# B&R Automation Studio project Servo
Automation Studio 4.12.2.93; technology packages: mappMotion 5.23.1, mappView 5.23.0

## Configuration Config1

CPU X20CP1586, AutomationRuntime B4.93, Build 4.1.2, Vc V4.72.6

### Task classes (Cpu.sw)
```
Cyclic#1 (cycle 8000 us, tolerance 0 us):
  servo <- servo.prg
DataObjects: McAcpSys
NcDataObjects: McDriveLog
Binaries: FWRules, McAcpSim, arcoal, arsvcreg, TCData, McAcpDrv, arflatprv, udbdef, iomap, Config_1, ashwd, arconfig, asfw, ashwac, sysconf, User, Role
Libraries: McBase, MpAxis, McAxis, MpBase, McAcpAx, fileio, powerlnk, sys_lib, asieccon, asepl, standard, MpAlarmX, astime, runtime
```

### Hardware
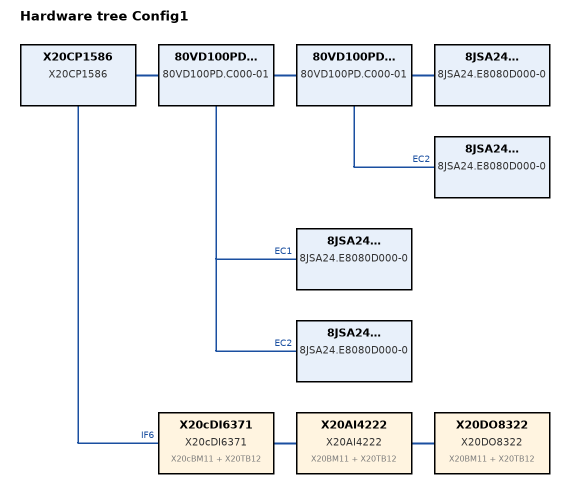
```
80VD100PD.C000-01 : 80VD100PD.C000-01 v2.5.0.0  [PLK1 -> 80VD100PD.C000-01a.PLK2 (NodeNumber=2) [Cable Type=PowerlinkCable, Length=10, Version=1.0.0.3]; EC1 -> 8JSA24.E8080D000-0.EC; EC2 -> 8JSA24.E8080D000-0a.EC; MT2 -> 8JSA24.E8080D000-0a.MT]
  DriveConfiguration/Module:
    McAcoposTypeID = AcoposMicroDConfig
    ActivateACOPOSSimulationOnPLC = 1
  DriveConfiguration/Channel[1]/RealAxis:
    AxisReference = gAxis_1
    MechanicalElementsIsInvisible = 0
  DriveConfiguration/Channel[1]/RealAxis/MechanicalElements/Gearbox:
    InputIsReadOnly = 0
    Input = 1
    OutputIsReadOnly = 0
    Output = 1
  DriveConfiguration/Channel[1]/RealAxis/MechanicalElements/RotaryToLinearTransformation:
    ReferenceDistanceIsReadOnly = 0
    ReferenceDistance = 1
  DriveConfiguration/Channel[1]/RealAxis/Controller:
    ModeIsReadOnly = 0
    Mode = PositionController
  DriveConfiguration/Channel[1]/RealAxis/Controller/Mode/Position:
    ProportionalGain = 50.0
    IntegrationTime = 0.0
    PredictionTime = 0.0004
    TotalDelayTime = 0.0004
  DriveConfiguration/Channel[1]/RealAxis/Controller/Mode/Speed:
    ProportionalGainIsReadOnly = 0
    ProportionalGain = 2.0
    IntegrationTimeIsReadOnly = 0
    IntegrationTime = 0.0
    FilterTimeIsReadOnly = 0
    FilterTime = 0.0
  DriveConfiguration/Channel[1]/RealAxis/Controller/Mode/LoopFilters:
    LoopFilterXIsReadOnly = 0
    LoopFilter1 = NotUsed
    LoopFilter2 = NotUsed
    LoopFilter3 = NotUsed
  DriveConfiguration/Channel[1]/RealAxis/Homing:
    ModeIsReadOnly = 0
    Mode = Direct
  DriveConfiguration/Channel[1]/RealAxis/Homing/Mode:
    Position = 0.0
    ReferencePulse = NotUsed
  DriveConfiguration/Channel[1]/RealAxis/Homing:
    RestorePositionVariable = 
  DriveConfiguration/Channel[1]/RealAxis/StopReaction:
    QuickstopIsReadOnly = 0
    Quickstop = DecelerationLimit
    DriveErrorIsReadOnly = 0
    DriveError = DecelerationLimit
  DriveConfiguration/Channel[1]/RealAxis/MovementErrorLimits:
    PositionError = 1.0
    VelocityErrorMonitoring = Automatic1
  DriveConfiguration/Channel[1]/RealAxis:
    JerkFilterIsReadOnly = 0
    JerkFilter = NotUsed
    ZeroVibrationFilter = NotUsed
  DriveConfiguration/Channel[1]/RealAxis/DigitalInputs/HomingSwitch:
    SourceIsReadOnly = 0
    Source = NotUsed
    Level = High
  DriveConfiguration/Channel[1]/RealAxis/DigitalInputs/PositiveLimitSwitch:
    SourceIsReadOnly = 0
    Source = NotUsed
    Level = High
  DriveConfiguration/Channel[1]/RealAxis/DigitalInputs/NegativeLimitSwitch:
    SourceIsReadOnly = 0
    Source = NotUsed
    Level = High
  DriveConfiguration/Channel[1]/RealAxis/DigitalInputs/Trigger1:
    Source = X2Trigger1
    Level = High
  DriveConfiguration/Channel[1]/RealAxis/DigitalInputs/Trigger2:
    Source = X2Trigger2
    Level = High
  DriveConfiguration/Channel[1]/RealAxis/DigitalInputs/Quickstop:
    Input = Trigger2
  DriveConfiguration/Channel[1]/RealAxis/Simulation:
    SimulationModeOnPLC = SetValueGeneration
    SimulationModeOnACOPOS = NotUsed
  DriveConfiguration/Channel[2]/RealAxis:
    AxisReference = gAxis_2
    MechanicalElementsIsInvisible = 0
  DriveConfiguration/Channel[2]/RealAxis/MechanicalElements/Gearbox:
    InputIsReadOnly = 0
    Input = 1
    OutputIsReadOnly = 0
    Output = 1
  DriveConfiguration/Channel[2]/RealAxis/MechanicalElements/RotaryToLinearTransformation:
    ReferenceDistanceIsReadOnly = 0
    ReferenceDistance = 1
  DriveConfiguration/Channel[2]/RealAxis/Controller:
    ModeIsReadOnly = 0
    Mode = PositionController
  DriveConfiguration/Channel[2]/RealAxis/Controller/Mode/Position:
    ProportionalGain = 50.0
    IntegrationTime = 0.0
    PredictionTime = 0.0004
    TotalDelayTime = 0.0004
  DriveConfiguration/Channel[2]/RealAxis/Controller/Mode/Speed:
    ProportionalGainIsReadOnly = 0
    ProportionalGain = 2.0
    IntegrationTimeIsReadOnly = 0
    IntegrationTime = 0.0
    FilterTimeIsReadOnly = 0
    FilterTime = 0.0
  DriveConfiguration/Channel[2]/RealAxis/Controller/Mode/LoopFilters:
    LoopFilterXIsReadOnly = 0
    LoopFilter1 = NotUsed
    LoopFilter2 = NotUsed
    LoopFilter3 = NotUsed
  DriveConfiguration/Channel[2]/RealAxis/Homing:
    ModeIsReadOnly = 0
    Mode = Direct
  DriveConfiguration/Channel[2]/RealAxis/Homing/Mode:
    Position = 0.0
    ReferencePulse = NotUsed
  DriveConfiguration/Channel[2]/RealAxis/Homing:
    RestorePositionVariable = 
  DriveConfiguration/Channel[2]/RealAxis/StopReaction:
    QuickstopIsReadOnly = 0
    Quickstop = DecelerationLimit
    DriveErrorIsReadOnly = 0
    DriveError = DecelerationLimit
  DriveConfiguration/Channel[2]/RealAxis/MovementErrorLimits:
    PositionError = 1.0
    VelocityErrorMonitoring = Automatic1
  DriveConfiguration/Channel[2]/RealAxis:
    JerkFilterIsReadOnly = 0
    JerkFilter = NotUsed
    ZeroVibrationFilter = NotUsed
  DriveConfiguration/Channel[2]/RealAxis/DigitalInputs/HomingSwitch:
    SourceIsReadOnly = 0
    Source = NotUsed
    Level = High
  DriveConfiguration/Channel[2]/RealAxis/DigitalInputs/PositiveLimitSwitch:
    SourceIsReadOnly = 0
    Source = NotUsed
    Level = High
  DriveConfiguration/Channel[2]/RealAxis/DigitalInputs/NegativeLimitSwitch:
    SourceIsReadOnly = 0
    Source = NotUsed
    Level = High
  DriveConfiguration/Channel[2]/RealAxis/DigitalInputs/Trigger1:
    Source = X2Trigger1
    Level = High
  DriveConfiguration/Channel[2]/RealAxis/DigitalInputs/Trigger2:
    Source = X2Trigger2
    Level = High
  DriveConfiguration/Channel[2]/RealAxis/DigitalInputs/Quickstop:
    Input = Trigger2
  DriveConfiguration/Channel[2]/RealAxis/Simulation:
    SimulationModeOnPLC = SetValueGeneration
    SimulationModeOnACOPOS = NotUsed
80VD100PD.C000-01a : 80VD100PD.C000-01 v2.5.0.0  [PLK1 -> X20CP1586.IF3 (NodeNumber=3) [Cable Type=PowerlinkCable, Length=10, Version=1.0.0.3]; PLK2 -> 80VD100PD.C000-01.PLK1 (NodeNumber=3) [Cable Type=PowerlinkCable, Length=10, Version=1.0.0.3]; EC1 -> 8JSA24.E8080D000-0b.EC; EC2 -> 8JSA24.E8080D000-0c.EC; MT2 -> 8JSA24.E8080D000-0c.MT]
  DriveConfiguration/Module:
    McAcoposTypeID = AcoposMicroDConfig
    ActivateACOPOSSimulationOnPLC = 1
  DriveConfiguration/Channel[1]/RealAxis:
    AxisReference = gAxis_3
    MechanicalElementsIsInvisible = 0
  DriveConfiguration/Channel[1]/RealAxis/MechanicalElements/Gearbox:
    InputIsReadOnly = 0
    Input = 1
    OutputIsReadOnly = 0
    Output = 1
  DriveConfiguration/Channel[1]/RealAxis/MechanicalElements/RotaryToLinearTransformation:
    ReferenceDistanceIsReadOnly = 0
    ReferenceDistance = 1
  DriveConfiguration/Channel[1]/RealAxis/Controller:
    ModeIsReadOnly = 0
    Mode = PositionController
  DriveConfiguration/Channel[1]/RealAxis/Controller/Mode/Position:
    ProportionalGain = 50.0
    IntegrationTime = 0.0
    PredictionTime = 0.0004
    TotalDelayTime = 0.0004
  DriveConfiguration/Channel[1]/RealAxis/Controller/Mode/Speed:
    ProportionalGainIsReadOnly = 0
    ProportionalGain = 2.0
    IntegrationTimeIsReadOnly = 0
    IntegrationTime = 0.0
    FilterTimeIsReadOnly = 0
    FilterTime = 0.0
  DriveConfiguration/Channel[1]/RealAxis/Controller/Mode/LoopFilters:
    LoopFilterXIsReadOnly = 0
    LoopFilter1 = NotUsed
    LoopFilter2 = NotUsed
    LoopFilter3 = NotUsed
  DriveConfiguration/Channel[1]/RealAxis/Homing:
    ModeIsReadOnly = 0
    Mode = Direct
  DriveConfiguration/Channel[1]/RealAxis/Homing/Mode:
    Position = 0.0
    ReferencePulse = Used
  DriveConfiguration/Channel[1]/RealAxis/Homing/Mode/ReferencePulse:
    HomingVelocity = 0.5
    Acceleration = 50.0
    HomingDirection = Positive
    KeepDirection = No
    ReferencePulseBlockingDistance = 0.0
  DriveConfiguration/Channel[1]/RealAxis/Homing:
    RestorePositionVariable = 
  DriveConfiguration/Channel[1]/RealAxis/StopReaction:
    QuickstopIsReadOnly = 0
    Quickstop = DecelerationLimit
    DriveErrorIsReadOnly = 0
    DriveError = DecelerationLimit
  DriveConfiguration/Channel[1]/RealAxis/MovementErrorLimits:
    PositionError = 1.0
    VelocityErrorMonitoring = Automatic1
  DriveConfiguration/Channel[1]/RealAxis:
    JerkFilterIsReadOnly = 0
    JerkFilter = NotUsed
    ZeroVibrationFilter = NotUsed
  DriveConfiguration/Channel[1]/RealAxis/DigitalInputs/HomingSwitch:
    SourceIsReadOnly = 0
    Source = NotUsed
    Level = High
  DriveConfiguration/Channel[1]/RealAxis/DigitalInputs/PositiveLimitSwitch:
    SourceIsReadOnly = 0
    Source = NotUsed
    Level = High
  DriveConfiguration/Channel[1]/RealAxis/DigitalInputs/NegativeLimitSwitch:
    SourceIsReadOnly = 0
    Source = NotUsed
    Level = High
  DriveConfiguration/Channel[1]/RealAxis/DigitalInputs/Trigger1:
    Source = X2Trigger1
    Level = High
  DriveConfiguration/Channel[1]/RealAxis/DigitalInputs/Trigger2:
    Source = X2Trigger2
    Level = High
  DriveConfiguration/Channel[1]/RealAxis/DigitalInputs/Quickstop:
    Input = Trigger2
  DriveConfiguration/Channel[1]/RealAxis/Simulation:
    SimulationModeOnPLC = SetValueGeneration
    SimulationModeOnACOPOS = NotUsed
  DriveConfiguration/Channel[2]/RealAxis:
    AxisReference = gAxis_4
    MechanicalElementsIsInvisible = 0
  DriveConfiguration/Channel[2]/RealAxis/MechanicalElements/Gearbox:
    InputIsReadOnly = 0
    Input = 1
    OutputIsReadOnly = 0
    Output = 1
  DriveConfiguration/Channel[2]/RealAxis/MechanicalElements/RotaryToLinearTransformation:
    ReferenceDistanceIsReadOnly = 0
    ReferenceDistance = 1
  DriveConfiguration/Channel[2]/RealAxis/Controller:
    ModeIsReadOnly = 0
    Mode = PositionController
  DriveConfiguration/Channel[2]/RealAxis/Controller/Mode/Position:
    ProportionalGain = 50.0
    IntegrationTime = 0.0
    PredictionTime = 0.0004
    TotalDelayTime = 0.0004
  DriveConfiguration/Channel[2]/RealAxis/Controller/Mode/Speed:
    ProportionalGainIsReadOnly = 0
    ProportionalGain = 2.0
    IntegrationTimeIsReadOnly = 0
    IntegrationTime = 0.0
    FilterTimeIsReadOnly = 0
    FilterTime = 0.0
  DriveConfiguration/Channel[2]/RealAxis/Controller/Mode/LoopFilters:
    LoopFilterXIsReadOnly = 0
    LoopFilter1 = NotUsed
    LoopFilter2 = NotUsed
    LoopFilter3 = NotUsed
  DriveConfiguration/Channel[2]/RealAxis/Homing:
    ModeIsReadOnly = 0
    Mode = Direct
  DriveConfiguration/Channel[2]/RealAxis/Homing/Mode:
    Position = 0.0
    ReferencePulse = NotUsed
  DriveConfiguration/Channel[2]/RealAxis/Homing:
    RestorePositionVariable = 
  DriveConfiguration/Channel[2]/RealAxis/StopReaction:
    QuickstopIsReadOnly = 0
    Quickstop = DecelerationLimit
    DriveErrorIsReadOnly = 0
    DriveError = DecelerationLimit
  DriveConfiguration/Channel[2]/RealAxis/MovementErrorLimits:
    PositionError = 1.0
    VelocityErrorMonitoring = Automatic1
  DriveConfiguration/Channel[2]/RealAxis:
    JerkFilterIsReadOnly = 0
    JerkFilter = NotUsed
    ZeroVibrationFilter = NotUsed
  DriveConfiguration/Channel[2]/RealAxis/DigitalInputs/HomingSwitch:
    SourceIsReadOnly = 0
    Source = NotUsed
    Level = High
  DriveConfiguration/Channel[2]/RealAxis/DigitalInputs/PositiveLimitSwitch:
    SourceIsReadOnly = 0
    Source = NotUsed
    Level = High
  DriveConfiguration/Channel[2]/RealAxis/DigitalInputs/NegativeLimitSwitch:
    SourceIsReadOnly = 0
    Source = NotUsed
    Level = High
  DriveConfiguration/Channel[2]/RealAxis/DigitalInputs/Trigger1:
    Source = X2Trigger1
    Level = High
  DriveConfiguration/Channel[2]/RealAxis/DigitalInputs/Trigger2:
    Source = X2Trigger2
    Level = High
  DriveConfiguration/Channel[2]/RealAxis/DigitalInputs/Quickstop:
    Input = Trigger2
  DriveConfiguration/Channel[2]/RealAxis/Simulation:
    SimulationModeOnPLC = SetValueGeneration
    SimulationModeOnACOPOS = NotUsed
8JSA24.E8080D000-0 : 8JSA24.E8080D000-0 v1.0.6.30  [EC -> 80VD100PD.C000-01.EC1; MT -> 80VD100PD.C000-01.MT1]
8JSA24.E8080D000-0a : 8JSA24.E8080D000-0 v1.0.6.30  [EC -> 80VD100PD.C000-01.EC2; MT -> 80VD100PD.C000-01.MT2]
8JSA24.E8080D000-0b : 8JSA24.E8080D000-0 v1.0.6.30  [EC -> 80VD100PD.C000-01a.EC1; MT -> 80VD100PD.C000-01a.MT1]
8JSA24.E8080D000-0c : 8JSA24.E8080D000-0 v1.0.6.30  [EC -> 80VD100PD.C000-01a.EC2; MT -> 80VD100PD.C000-01a.MT2]
X20AI4222 : X20AI4222 v1.2.0.0  [SS1 -> X20TB12b.SS; SL -> X20BM11a.SL1]
X20BM11 : X20BM11 v1.1.0.0  [X2X1 -> X20BM11a.X2X2]
X20BM11a : X20BM11 v1.1.0.0  [X2X1 -> X20cBM11.X2X2]
X20CP1586 : X20CP1586 v1.10.0.0
  Connector IF2:
    ActivateDevice = 1
  ConfigurationID = Servo_Config1
  Simulation = 1
  TimerDeviceType = EPLX2X
  TimerDevice = X20CP1586.IF3
  TaskClassIdleTime = 2000
  Cyclic1Duration = 8000
  Cyclic1Tolerance = 0
  Cyclic1Stack = 35563
  FileDevice1
  FileDeviceName1 = USER
  FileDevicePath1 = USER_PATH
  ActivateOpcUa = 1
  OpcUaInformationModels_PV_Version = 1
X20DO8322 : X20DO8322 v1.5.0.0  [SS1 -> X20TB12a.SS; SL -> X20BM11.SL1]
X20TB12 : X20TB12 v1.0.0.0
X20TB12a : X20TB12 v1.0.0.0
X20TB12b : X20TB12 v1.0.0.0
X20cBM11 : X20cBM11 v1.1.0.0  [X2X1 -> X20CP1586.IF6]
X20cDI6371 : X20cDI6371 v1.2.0.0  [SS1 -> X20TB12.SS; SL -> X20cBM11.SL1]
```

### IoMap.iom - X20CP1586/IoMap.iom
```iecst
VAR_CONFIG
	::KEY AT %IX."X20cDI6371".DigitalInput01;
	::Left_Proximity AT %IX."X20cDI6371".DigitalInput03;
	::Buzzer AT %QX."X20DO8322".DigitalOutput01;
	::LeftAct AT %QX."X20DO8322".DigitalOutput02;
	::RightAct AT %QX."X20DO8322".DigitalOutput03;
	::Proximity_1 AT %IX."X20cDI6371".DigitalInput02;
	::Right_Proximity AT %IX."X20cDI6371".DigitalInput04;
END_VAR
```

### Config_1.axis - X20CP1586/mappMotion/Config_1.axis
```
Element gAxis_1 (Type=axis)
  BaseTypeIsReadOnly = 0
  BaseType = LinearBounded
    MeasurementUnit = 5066068
    MeasurementResolutionIsReadOnly = 0
    MeasurementResolution = 0.01
    CountDirectionIsReadOnly = 0
    CountDirection = Standard
  MovementLimitsIsReadOnly = 0
  MovementLimits = Internal
    Position:
      LowerLimitMin = -1.79769313486231E308
      UpperLimitMax = 1.79769313486231E308
      LowerLimit = -100000
      UpperLimit = 100000
    VelocityIsReadOnly = 0
    Velocity:
      VelocityMax = 3.4E38
      Velocity = 10
    AccelerationIsReadOnly = 0
    Acceleration:
      AccelerationMax = 3.4E38
      Acceleration = 50
    DecelerationIsReadOnly = 0
    Deceleration:
      DecelerationMax = 3.4E38
      Deceleration = 50.0
  Alarms = None
```

### Config_2.axis - X20CP1586/mappMotion/Config_2.axis
```
Element gAxis_2 (Type=axis)
  BaseTypeIsReadOnly = 0
  BaseType = LinearBounded
    MeasurementUnit = 5066068
    MeasurementResolutionIsReadOnly = 0
    MeasurementResolution = 0.01
    CountDirectionIsReadOnly = 0
    CountDirection = Standard
  MovementLimitsIsReadOnly = 0
  MovementLimits = Internal
    Position:
      LowerLimitMin = -1.79769313486231E308
      UpperLimitMax = 1.79769313486231E308
      LowerLimit = -1000.0
      UpperLimit = 1000.0
    VelocityIsReadOnly = 0
    Velocity:
      VelocityMax = 3.4E38
      Velocity = 10.0
    AccelerationIsReadOnly = 0
    Acceleration:
      AccelerationMax = 3.4E38
      Acceleration = 50.0
    DecelerationIsReadOnly = 0
    Deceleration:
      DecelerationMax = 3.4E38
      Deceleration = 50.0
  Alarms = None
```

### Config_3.axis - X20CP1586/mappMotion/Config_3.axis
```
Element gAxis_3 (Type=axis)
  BaseTypeIsReadOnly = 0
  BaseType = LinearBounded
    MeasurementUnit = 5066068
    MeasurementResolutionIsReadOnly = 0
    MeasurementResolution = 0.01
    CountDirectionIsReadOnly = 0
    CountDirection = Standard
  MovementLimitsIsReadOnly = 0
  MovementLimits = Internal
    Position:
      LowerLimitMin = -1.79769313486231E308
      UpperLimitMax = 1.79769313486231E308
      LowerLimit = -1000.0
      UpperLimit = 1000.0
    VelocityIsReadOnly = 0
    Velocity:
      VelocityMax = 3.4E38
      Velocity = 10.0
    AccelerationIsReadOnly = 0
    Acceleration:
      AccelerationMax = 3.4E38
      Acceleration = 50.0
    DecelerationIsReadOnly = 0
    Deceleration:
      DecelerationMax = 3.4E38
      Deceleration = 50.0
  Alarms = None
```

### Config_4.axis - X20CP1586/mappMotion/Config_4.axis
```
Element gAxis_4 (Type=axis)
  BaseTypeIsReadOnly = 0
  BaseType = LinearBounded
    MeasurementUnit = 5066068
    MeasurementResolutionIsReadOnly = 0
    MeasurementResolution = 0.01
    CountDirectionIsReadOnly = 0
    CountDirection = Standard
  MovementLimitsIsReadOnly = 0
  MovementLimits = Internal
    Position:
      LowerLimitMin = -1.79769313486231E308
      UpperLimitMax = 1.79769313486231E308
      LowerLimit = -1000.0
      UpperLimit = 1000.0
    VelocityIsReadOnly = 0
    Velocity:
      VelocityMax = 3.4E38
      Velocity = 10.0
    AccelerationIsReadOnly = 0
    Acceleration:
      AccelerationMax = 3.4E38
      Acceleration = 50.0
    DecelerationIsReadOnly = 0
    Deceleration:
      DecelerationMax = 3.4E38
      Deceleration = 50.0
  Alarms = None
```

### Config.mpalarmxcore - X20CP1586/mappServices/Config.mpalarmxcore
```
Element gAlarmXCore (Type=mpalarmxcore)
  mapp.AlarmX.Core.Configuration:
    [0]:
      Name = Full
      Message = Herbicide solution Full
      Code = 101
      Severity = 3001
      Behavior = PersistentAlarm
    [1]:
      Name = Low
      Message = Herbicide solution in Half
      Code = 102
      Severity = 3002
      Behavior = PersistentAlarm
    [2]:
      Name = Very Low
      Message = Herbicide solution is low
      Code = 103
      Severity = 3003
      Behavior = PersistentAlarm
```

### Config_5.mpalarmxhistory - X20CP1586/mappServices/Config_5.mpalarmxhistory
```
Element gAlarmXHistory (Type=mpalarmxhistory)
  mapp.AlarmX.History.Queries:
    [0]:
      Name = WeedicideMedium
```

## Logical view

Binary libraries used (declarations not repeated): operator, runtime, astime, AsIecCon, McBase, MpAxis, McAxis, MpBase, McAcpAx, standard

### Global.var - Global variables
```iecst
VAR
	RightAct : BOOL;
	Left_Proximity : BOOL;
	Right_Solenoid : BOOL;
	KEY : BOOL;
	Buzzer : BOOL;
	Right_Proximity : BOOL;
	Left_Solenoid : BOOL;
	LeftAct : BOOL;
	Proximity_1 : BOOL;
	Counter : INT := 0;
	Row : INT;
	LeftWheel_F : MpAxisBasic;
	LeftWheel_B : MpAxisBasic;
	RightWheel_F : MpAxisBasic;
	RightWheel_B : MpAxisBasic;
	AxisParameters : MpAxisBasicParType;
	Float_2 : BOOL;
	Float_1 : BOOL;
	FloatSensor : INT;
	State : BOOL := FALSE;
	Pump : BOOL := TRUE;
END_VAR
```


### Program Logical/servo (IEC)

#### Variables.var
```iecst
VAR
	TON_0 : TON;
	TON_1 : TON;
END_VAR
```

#### Main.st
```iecst
PROGRAM _INIT
	LeftWheel_F.Enable := TRUE;
	LeftWheel_F.MpLink := ADR(gAxis_1);
	LeftWheel_F.Parameters := ADR(AxisParameters);

	LeftWheel_B.Enable := TRUE;
	LeftWheel_B.MpLink := ADR(gAxis_2);
	LeftWheel_B.Parameters := ADR(AxisParameters);

	RightWheel_F.Enable := TRUE;
	RightWheel_F.MpLink := ADR(gAxis_3);
	RightWheel_F.Parameters := ADR(AxisParameters);

	RightWheel_B.Enable := TRUE;
	RightWheel_B.MpLink := ADR(gAxis_4);
	RightWheel_B.Parameters := ADR(AxisParameters);
END_PROGRAM

PROGRAM _CYCLIC
	//Front LeftWheel Ingnition
	IF LeftWheel_F.Info.ReadyToPowerOn = TRUE THEN
		LeftWheel_F.Power := TRUE;
	END_IF
	IF LeftWheel_F.PowerOn = TRUE THEN
		LeftWheel_F.Home := TRUE;
	END_IF
	IF LeftWheel_F.IsHomed = TRUE THEN
		LeftWheel_F.MoveVelocity := TRUE;
	END_IF
	//Back LeftWheel Ingnition
	IF LeftWheel_F.Info.ReadyToPowerOn = TRUE THEN
		LeftWheel_F.Power := TRUE;
	END_IF
	IF LeftWheel_F.PowerOn = TRUE THEN
		LeftWheel_F.Home := TRUE;
	END_IF
	IF LeftWheel_F.IsHomed = TRUE THEN
		LeftWheel_F.MoveVelocity := TRUE;
	END_IF
	//Front RightWheel Ingnition
	IF LeftWheel_F.Info.ReadyToPowerOn = TRUE THEN
		LeftWheel_F.Power := TRUE;
	END_IF
	IF LeftWheel_F.PowerOn = TRUE THEN
		LeftWheel_F.Home := TRUE;
	END_IF
	IF LeftWheel_F.IsHomed = TRUE THEN
		LeftWheel_F.MoveVelocity := TRUE;
	END_IF
	//Back RightWheel Ingnition
	IF LeftWheel_F.Info.ReadyToPowerOn = TRUE THEN
		LeftWheel_F.Power := TRUE;
	END_IF
	IF LeftWheel_F.PowerOn = TRUE THEN
		LeftWheel_F.Home := TRUE;
	END_IF

	IF LeftWheel_F.IsHomed = TRUE THEN
		LeftWheel_F.MoveVelocity := TRUE;
	END_IF

	(*LeftWheel_F.MoveVelocity := TRUE;
	LeftWheel_B.MoveVelocity := TRUE;
	RightWheel_F.MoveVelocity := TRUE;
	RightWheel_B.MoveVelocity := TRUE;*)

	//Robot Identification
	IF KEY = TRUE THEN
		Buzzer := TRUE;
	ELSE
		Buzzer := FALSE;
	END_IF

	//Robot Turning
	IF Proximity_1 = 1 AND NOT State THEN
		Counter := Counter+1;
		Pump := FALSE;
		Row := Counter MOD 2;
		State := Proximity_1;
		(*IF Row = 0 THEN
			LeftWheel_F.MpLink := ADR(gAxis_1);
			LeftWheel_F.MoveVelocity := FALSE;
			LeftWheel_F.Parameters := ADR(AxisParameters);
			LeftWheel_F();

			LeftWheel_B.MpLink := ADR(gAxis_2);
			LeftWheel_B.MoveVelocity := FALSE;
			LeftWheel_B.Parameters := ADR(AxisParameters);
			LeftWheel_B();

		ELSE

			RightWheel_F.MpLink := ADR(gAxis_3);
			RightWheel_F.MoveVelocity := FALSE;
			RightWheel_F.Parameters := ADR(AxisParameters);
			RightWheel_F();

			RightWheel_B.MpLink := ADR(gAxis_4);
			RightWheel_B.MoveVelocity := FALSE;
			RightWheel_B.Parameters := ADR(AxisParameters);
			RightWheel_B();
		END_IF*)
	END_IF
	//Left Sensor
	IF Right_Proximity = 1 THEN
		Right_Solenoid := FALSE;
		RightAct := TRUE;
	ELSE
		Right_Solenoid := TRUE;
		RightAct := FALSE;
	END_IF

	//Right Sensor
	IF Left_Proximity = 1 THEN
		Left_Solenoid := FALSE;
		LeftAct := TRUE;
	ELSE
		Left_Solenoid := TRUE;
		LeftAct := FALSE;
	END_IF

	//Floatsensor value Float1 Float2
	IF 	FloatSensor<3 AND FloatSensor>1 THEN
		Float_1:=TRUE;
		Float_2:=FALSE;
	ELSIF FloatSensor<1 THEN
		Float_2:=TRUE;
		Float_1:=TRUE;
	ELSE
		Float_1:=FALSE;
		Float_2:=FALSE;
	END_IF;

	LeftWheel_F();
	LeftWheel_B();
	RightWheel_F();
	RightWheel_B();
	END_PROGRAM

PROGRAM _EXIT
	(*LeftWheel_F.Power  := FALSE;
	LeftWheel_F.Home   := FALSE;
	LeftWheel_F.MoveAbsolute := FALSE;
	LeftWheel_F.MoveAdditive := FALSE;
	LeftWheel_F.MoveVelocity := FALSE;
	LeftWheel_F.Stop         := FALSE;
	LeftWheel_F.ErrorReset   := FALSE;
	LeftWheel_F();*)
END_PROGRAM
```

- Visualisation Logical/mappView (not shown)

Listed in the project but not available here: Logical/Global.typ
